PROGRAM VariablePersistence
VAR
	fbCX565304_PER :FB_S_UPS_CX51x0;
END_VAR


//Save Peristent Data 
fbCX565304_PER(
	sNetID:= , //'5.86.83.4.4.1'
	iPLCPort:= 851, 
	tTimeout:= DEFAULT_ADS_TIMEOUT, 
	eUpsMode:= eSUPS_WrPersistData_NoShutdown, 
	ePersistentMode:= SPDM_2PASS, 
	tRecoverTime:= T#10S, 
	bPowerFailDetect=> , 
	eState=> );

END_PROGRAM

(* stored: Version 1.1.0.1, ProductVersion 3.1.4024.9
   POU VariablePersistence: Id {7495d68e-5062-4f43-bcb1-46f6e9da2a9c}, SpecialFunc None *)
